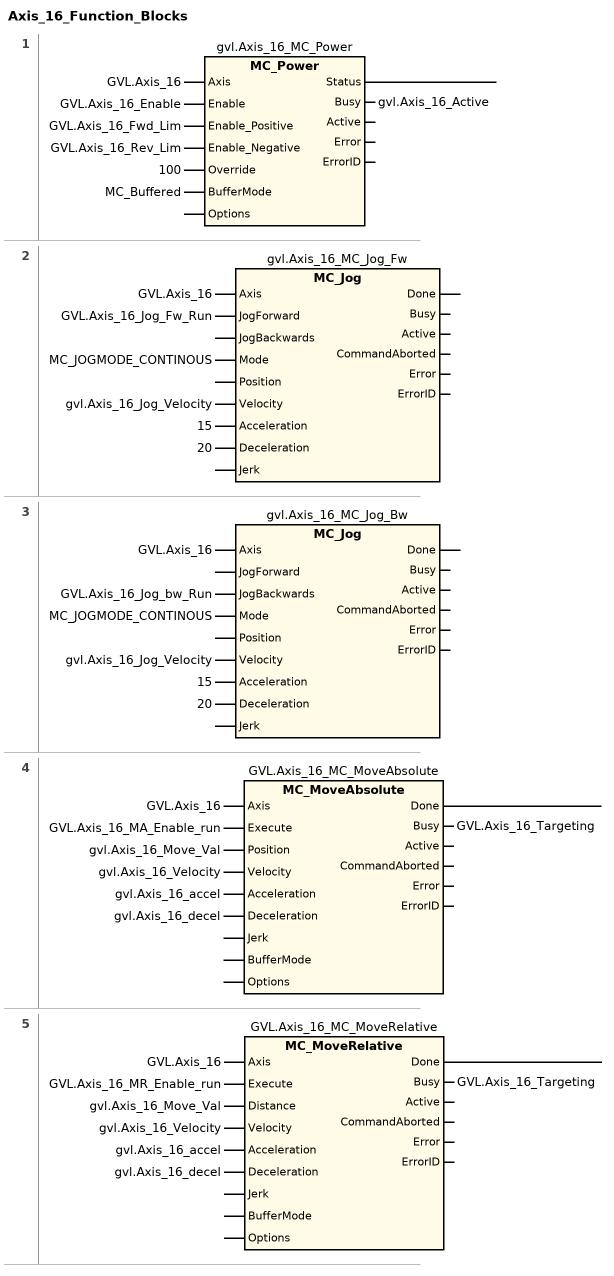
// NETWORK 1
gvl.Axis_16_MC_Power(
    Axis := GVL.Axis_16,
    Enable := GVL.Axis_16_Enable,
    Enable_Positive := GVL.Axis_16_Fwd_Lim,
    Enable_Negative := GVL.Axis_16_Rev_Lim,
    Override := 100,
    BufferMode := MC_Buffered,
    Busy => gvl.Axis_16_Active); // MC_Power

// NETWORK 2
gvl.Axis_16_MC_Jog_Fw(
    Axis := GVL.Axis_16,
    JogForward := GVL.Axis_16_Jog_Fw_Run,
    Mode := MC_JOGMODE_CONTINOUS,
    Velocity := gvl.Axis_16_Jog_Velocity,
    Acceleration := 15,
    Deceleration := 20); // MC_Jog

// NETWORK 3
gvl.Axis_16_MC_Jog_Bw(
    Axis := GVL.Axis_16,
    JogBackwards := GVL.Axis_16_Jog_bw_Run,
    Mode := MC_JOGMODE_CONTINOUS,
    Velocity := gvl.Axis_16_Jog_Velocity,
    Acceleration := 15,
    Deceleration := 20); // MC_Jog

// NETWORK 4
GVL.Axis_16_MC_MoveAbsolute(
    Axis := GVL.Axis_16,
    Execute := GVL.Axis_16_MA_Enable_run,
    Position := gvl.Axis_16_Move_Val,
    Velocity := gvl.Axis_16_Velocity,
    Acceleration := gvl.Axis_16_accel,
    Deceleration := gvl.Axis_16_decel,
    Busy => GVL.Axis_16_Targeting); // MC_MoveAbsolute

// NETWORK 5
GVL.Axis_16_MC_MoveRelative(
    Axis := GVL.Axis_16,
    Execute := GVL.Axis_16_MR_Enable_run,
    Distance := gvl.Axis_16_Move_Val,
    Velocity := gvl.Axis_16_Velocity,
    Acceleration := gvl.Axis_16_accel,
    Deceleration := gvl.Axis_16_decel,
    Busy => GVL.Axis_16_Targeting); // MC_MoveRelative

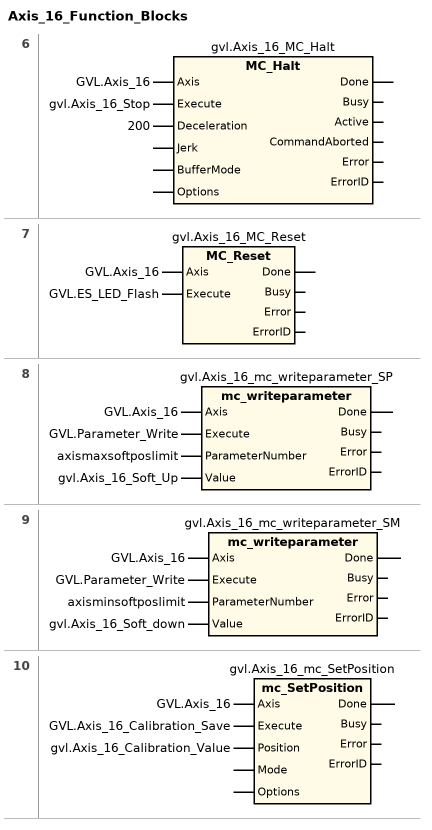
// NETWORK 6
gvl.Axis_16_MC_Halt(Axis := GVL.Axis_16, Execute := gvl.Axis_16_Stop, Deceleration := 200); // MC_Halt

// NETWORK 7
gvl.Axis_16_MC_Reset(Axis := GVL.Axis_16, Execute := GVL.ES_LED_Flash); // MC_Reset

// NETWORK 8
gvl.Axis_16_mc_writeparameter_SP(
    Axis := GVL.Axis_16,
    Execute := GVL.Parameter_Write,
    ParameterNumber := axismaxsoftposlimit,
    Value := gvl.Axis_16_Soft_Up); // mc_writeparameter

// NETWORK 9
gvl.Axis_16_mc_writeparameter_SM(
    Axis := GVL.Axis_16,
    Execute := GVL.Parameter_Write,
    ParameterNumber := axisminsoftposlimit,
    Value := gvl.Axis_16_Soft_down); // mc_writeparameter

// NETWORK 10
gvl.Axis_16_mc_SetPosition(
    Axis := GVL.Axis_16,
    Execute := GVL.Axis_16_Calibration_Save,
    Position := gvl.Axis_16_Calibration_Value); // mc_SetPosition

END_PROGRAM

// ---- POUs/Axis_16_Logic.TcPOU
PROGRAM Axis_16_Logic
VAR
	TON_0: TON;
	TON_1: TON;
	TON_2: TON;
	TON_3: TON;
	Axis_16_Velocity_Range: LREAL;
	Axis_16_Velocity_Scale: LREAL;
	Axis_16_Velocity_Raw: LREAL;
	Axis_16_Soft_Range: LREAL;
	Axis_16_Soft_Position: LREAL;
	Axis_16_Soft_Position_In_Range: LREAL;
END_VAR

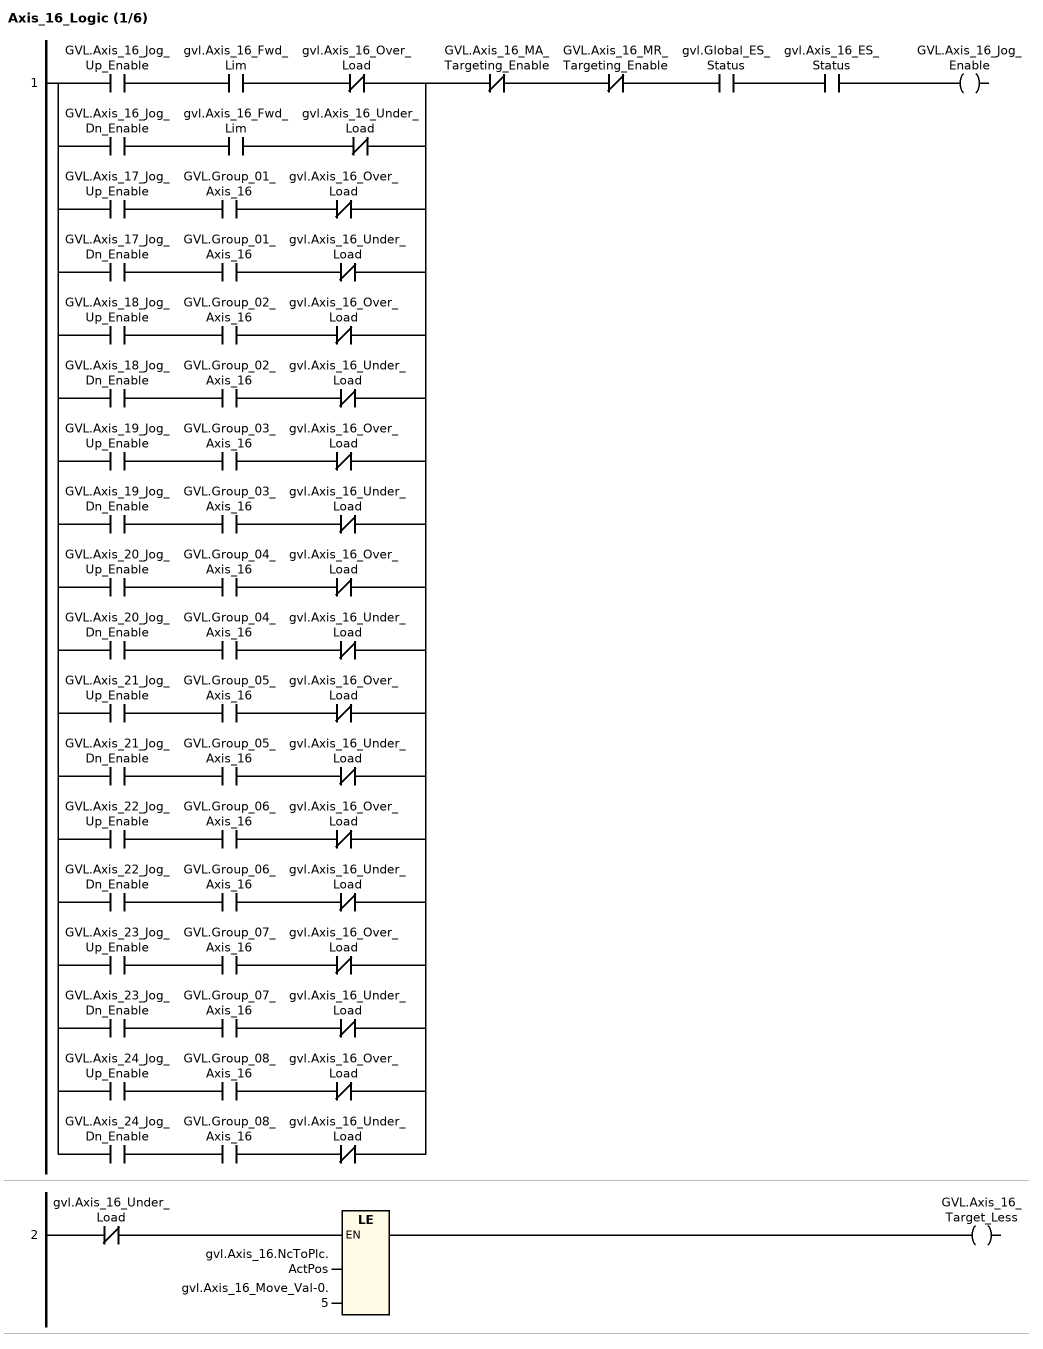
// NETWORK 1
GVL.Axis_16_Jog_Enable := (GVL.Axis_16_Jog_Up_Enable AND gvl.Axis_16_Fwd_Lim AND NOT gvl.Axis_16_Over_Load OR GVL.Axis_16_Jog_Dn_Enable AND gvl.Axis_16_Fwd_Lim AND NOT gvl.Axis_16_Under_Load OR GVL.Axis_17_Jog_Up_Enable AND GVL.Group_01_Axis_16 AND NOT gvl.Axis_16_Over_Load OR GVL.Axis_17_Jog_Dn_Enable AND GVL.Group_01_Axis_16 AND NOT gvl.Axis_16_Under_Load OR GVL.Axis_18_Jog_Up_Enable AND GVL.Group_02_Axis_16 AND NOT gvl.Axis_16_Over_Load OR GVL.Axis_18_Jog_Dn_Enable AND GVL.Group_02_Axis_16 AND NOT gvl.Axis_16_Under_Load OR GVL.Axis_19_Jog_Up_Enable AND GVL.Group_03_Axis_16 AND NOT gvl.Axis_16_Over_Load OR GVL.Axis_19_Jog_Dn_Enable AND GVL.Group_03_Axis_16 AND NOT gvl.Axis_16_Under_Load OR GVL.Axis_20_Jog_Up_Enable AND GVL.Group_04_Axis_16 AND NOT gvl.Axis_16_Over_Load OR GVL.Axis_20_Jog_Dn_Enable AND GVL.Group_04_Axis_16 AND NOT gvl.Axis_16_Under_Load OR GVL.Axis_21_Jog_Up_Enable AND GVL.Group_05_Axis_16 AND NOT gvl.Axis_16_Over_Load OR GVL.Axis_21_Jog_Dn_Enable AND GVL.Group_05_Axis_16 AND NOT gvl.Axis_16_Under_Load OR GVL.Axis_22_Jog_Up_Enable AND GVL.Group_06_Axis_16 AND NOT gvl.Axis_16_Over_Load OR GVL.Axis_22_Jog_Dn_Enable AND GVL.Group_06_Axis_16 AND NOT gvl.Axis_16_Under_Load OR GVL.Axis_23_Jog_Up_Enable AND GVL.Group_07_Axis_16 AND NOT gvl.Axis_16_Over_Load OR GVL.Axis_23_Jog_Dn_Enable AND GVL.Group_07_Axis_16 AND NOT gvl.Axis_16_Under_Load OR GVL.Axis_24_Jog_Up_Enable AND GVL.Group_08_Axis_16 AND NOT gvl.Axis_16_Over_Load OR GVL.Axis_24_Jog_Dn_Enable AND GVL.Group_08_Axis_16 AND NOT gvl.Axis_16_Under_Load) AND NOT GVL.Axis_16_MA_Targeting_Enable AND NOT GVL.Axis_16_MR_Targeting_Enable AND gvl.Global_ES_Status AND gvl.Axis_16_ES_Status;

// NETWORK 2
GVL.Axis_16_Target_Less := NOT gvl.Axis_16_Under_Load AND gvl.Axis_16.NcToPlc.ActPos <= (gvl.Axis_16_Move_Val-0.5);

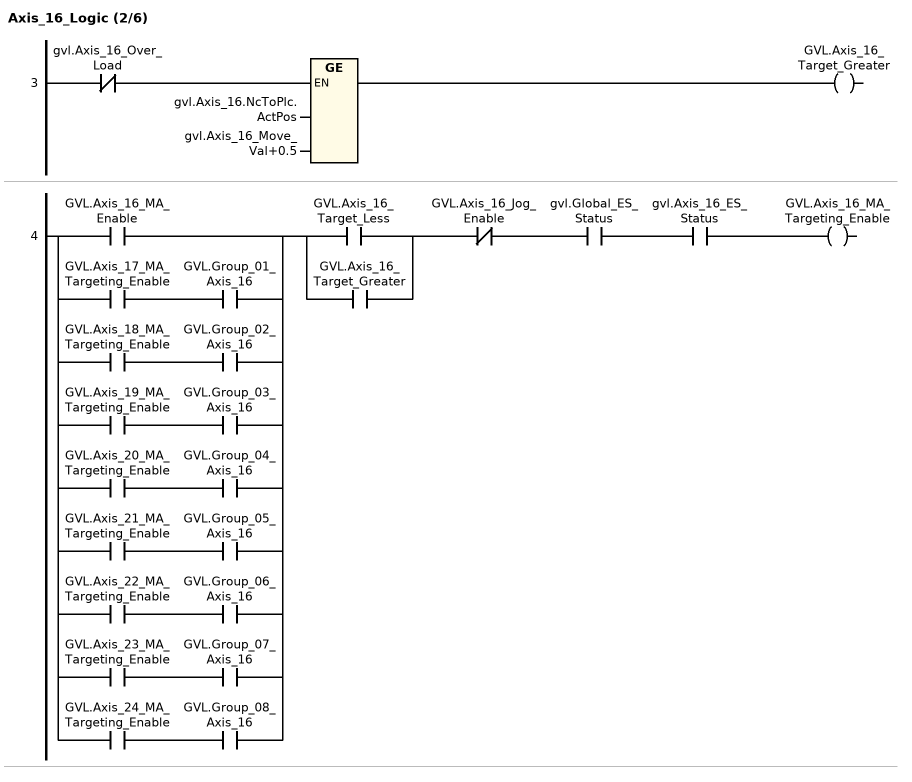
// NETWORK 3
GVL.Axis_16_Target_Greater := NOT gvl.Axis_16_Over_Load AND gvl.Axis_16.NcToPlc.ActPos >= (gvl.Axis_16_Move_Val+0.5);

// NETWORK 4
GVL.Axis_16_MA_Targeting_Enable := (GVL.Axis_16_MA_Enable OR GVL.Axis_17_MA_Targeting_Enable AND GVL.Group_01_Axis_16 OR GVL.Axis_18_MA_Targeting_Enable AND GVL.Group_02_Axis_16 OR GVL.Axis_19_MA_Targeting_Enable AND GVL.Group_03_Axis_16 OR GVL.Axis_20_MA_Targeting_Enable AND GVL.Group_04_Axis_16 OR GVL.Axis_21_MA_Targeting_Enable AND GVL.Group_05_Axis_16 OR GVL.Axis_22_MA_Targeting_Enable AND GVL.Group_06_Axis_16 OR GVL.Axis_23_MA_Targeting_Enable AND GVL.Group_07_Axis_16 OR GVL.Axis_24_MA_Targeting_Enable AND GVL.Group_08_Axis_16) AND (GVL.Axis_16_Target_Less OR GVL.Axis_16_Target_Greater) AND NOT GVL.Axis_16_Jog_Enable AND gvl.Global_ES_Status AND gvl.Axis_16_ES_Status;

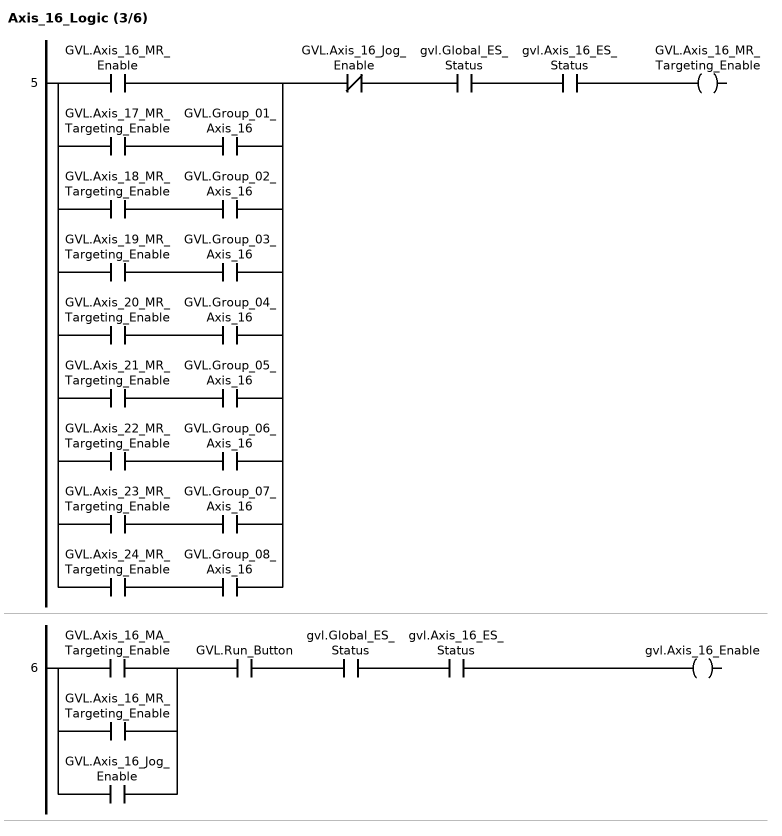
// NETWORK 5
GVL.Axis_16_MR_Targeting_Enable := (GVL.Axis_16_MR_Enable OR GVL.Axis_17_MR_Targeting_Enable AND GVL.Group_01_Axis_16 OR GVL.Axis_18_MR_Targeting_Enable AND GVL.Group_02_Axis_16 OR GVL.Axis_19_MR_Targeting_Enable AND GVL.Group_03_Axis_16 OR GVL.Axis_20_MR_Targeting_Enable AND GVL.Group_04_Axis_16 OR GVL.Axis_21_MR_Targeting_Enable AND GVL.Group_05_Axis_16 OR GVL.Axis_22_MR_Targeting_Enable AND GVL.Group_06_Axis_16 OR GVL.Axis_23_MR_Targeting_Enable AND GVL.Group_07_Axis_16 OR GVL.Axis_24_MR_Targeting_Enable AND GVL.Group_08_Axis_16) AND NOT GVL.Axis_16_Jog_Enable AND gvl.Global_ES_Status AND gvl.Axis_16_ES_Status;

// NETWORK 6
gvl.Axis_16_Enable := (GVL.Axis_16_MA_Targeting_Enable OR GVL.Axis_16_MR_Targeting_Enable OR GVL.Axis_16_Jog_Enable) AND GVL.Run_Button AND gvl.Global_ES_Status AND gvl.Axis_16_ES_Status;

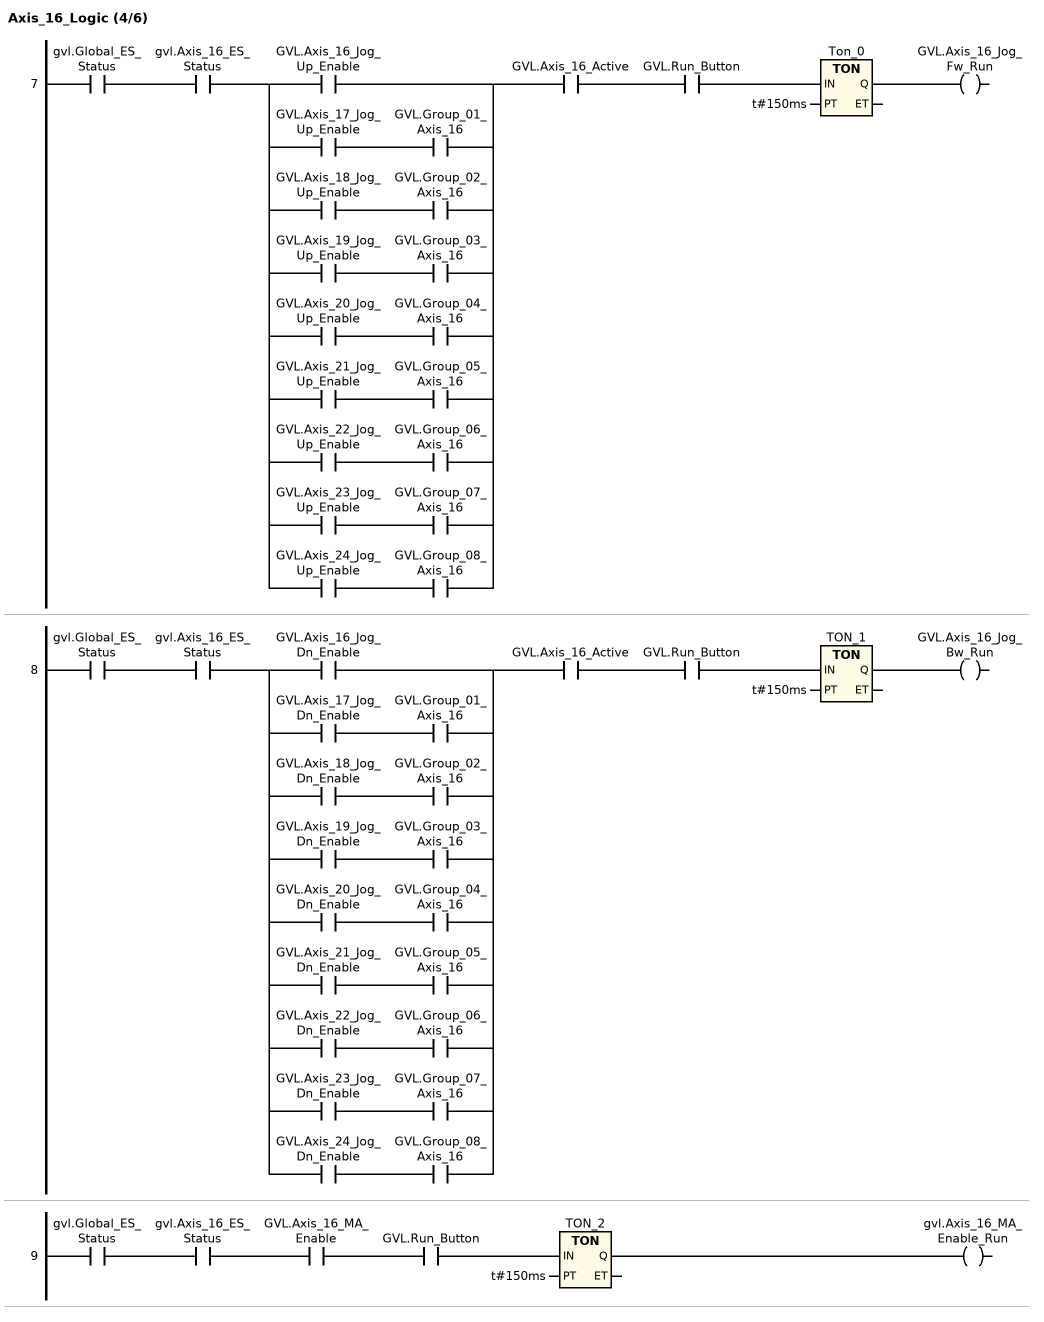
// NETWORK 7
Ton_0(IN := gvl.Global_ES_Status AND gvl.Axis_16_ES_Status AND (GVL.Axis_16_Jog_Up_Enable OR GVL.Axis_17_Jog_Up_Enable AND GVL.Group_01_Axis_16 OR GVL.Axis_18_Jog_Up_Enable AND GVL.Group_02_Axis_16 OR GVL.Axis_19_Jog_Up_Enable AND GVL.Group_03_Axis_16 OR GVL.Axis_20_Jog_Up_Enable AND GVL.Group_04_Axis_16 OR GVL.Axis_21_Jog_Up_Enable AND GVL.Group_05_Axis_16 OR GVL.Axis_22_Jog_Up_Enable AND GVL.Group_06_Axis_16 OR GVL.Axis_23_Jog_Up_Enable AND GVL.Group_07_Axis_16 OR GVL.Axis_24_Jog_Up_Enable AND GVL.Group_08_Axis_16) AND GVL.Axis_16_Active AND GVL.Run_Button, PT := t#150ms); // TON
GVL.Axis_16_Jog_Fw_Run := Ton_0.Q;

// NETWORK 8
TON_1(IN := gvl.Global_ES_Status AND gvl.Axis_16_ES_Status AND (GVL.Axis_16_Jog_Dn_Enable OR GVL.Axis_17_Jog_Dn_Enable AND GVL.Group_01_Axis_16 OR GVL.Axis_18_Jog_Dn_Enable AND GVL.Group_02_Axis_16 OR GVL.Axis_19_Jog_Dn_Enable AND GVL.Group_03_Axis_16 OR GVL.Axis_20_Jog_Dn_Enable AND GVL.Group_04_Axis_16 OR GVL.Axis_21_Jog_Dn_Enable AND GVL.Group_05_Axis_16 OR GVL.Axis_22_Jog_Dn_Enable AND GVL.Group_06_Axis_16 OR GVL.Axis_23_Jog_Dn_Enable AND GVL.Group_07_Axis_16 OR GVL.Axis_24_Jog_Dn_Enable AND GVL.Group_08_Axis_16) AND GVL.Axis_16_Active AND GVL.Run_Button, PT := t#150ms); // TON
GVL.Axis_16_Jog_Bw_Run := TON_1.Q;

// NETWORK 9
TON_2(IN := gvl.Global_ES_Status AND gvl.Axis_16_ES_Status AND GVL.Axis_16_MA_Enable AND GVL.Run_Button, PT := t#150ms); // TON
gvl.Axis_16_MA_Enable_Run := TON_2.Q;

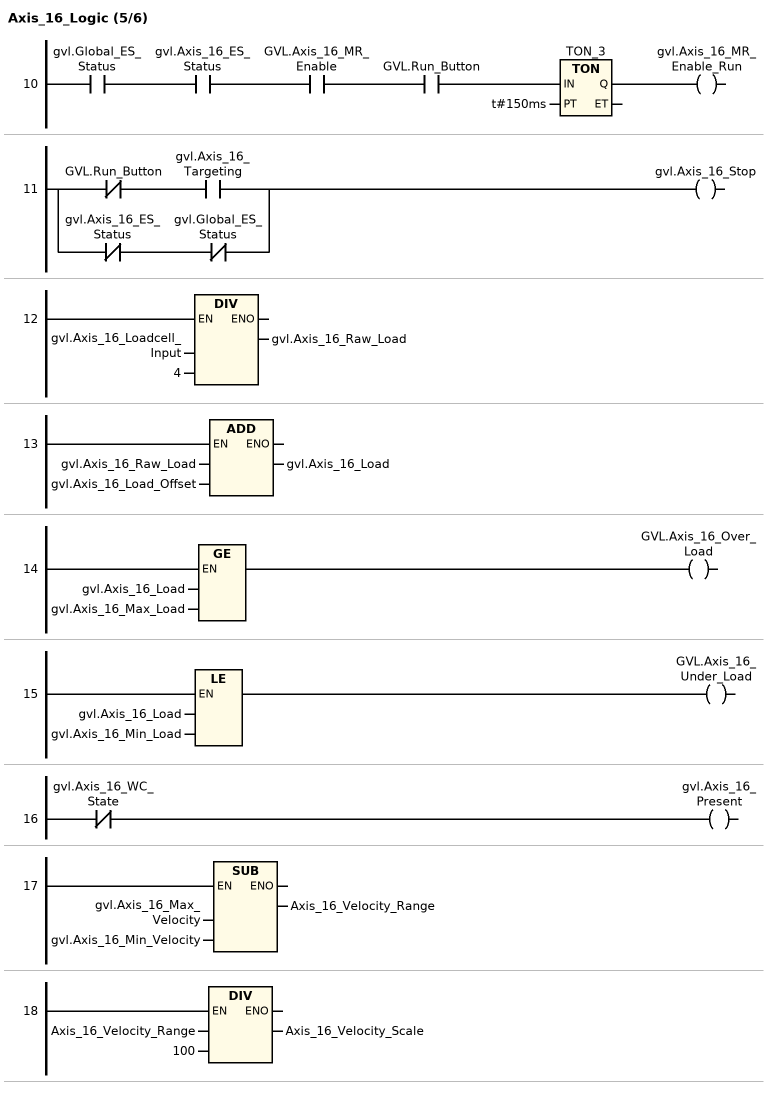
// NETWORK 10
TON_3(IN := gvl.Global_ES_Status AND gvl.Axis_16_ES_Status AND GVL.Axis_16_MR_Enable AND GVL.Run_Button, PT := t#150ms); // TON
gvl.Axis_16_MR_Enable_Run := TON_3.Q;

// NETWORK 11
gvl.Axis_16_Stop := NOT GVL.Run_Button AND gvl.Axis_16_Targeting OR NOT gvl.Axis_16_ES_Status AND NOT gvl.Global_ES_Status;

// NETWORK 12
gvl.Axis_16_Raw_Load := gvl.Axis_16_Loadcell_Input / 4;

// NETWORK 13
gvl.Axis_16_Load := gvl.Axis_16_Raw_Load + gvl.Axis_16_Load_Offset;

// NETWORK 14
GVL.Axis_16_Over_Load := gvl.Axis_16_Load >= gvl.Axis_16_Max_Load;

// NETWORK 15
GVL.Axis_16_Under_Load := gvl.Axis_16_Load <= gvl.Axis_16_Min_Load;

// NETWORK 16
gvl.Axis_16_Present := NOT gvl.Axis_16_WC_State;

// NETWORK 17
Axis_16_Velocity_Range := gvl.Axis_16_Max_Velocity - gvl.Axis_16_Min_Velocity;

// NETWORK 18
Axis_16_Velocity_Scale := Axis_16_Velocity_Range / 100;

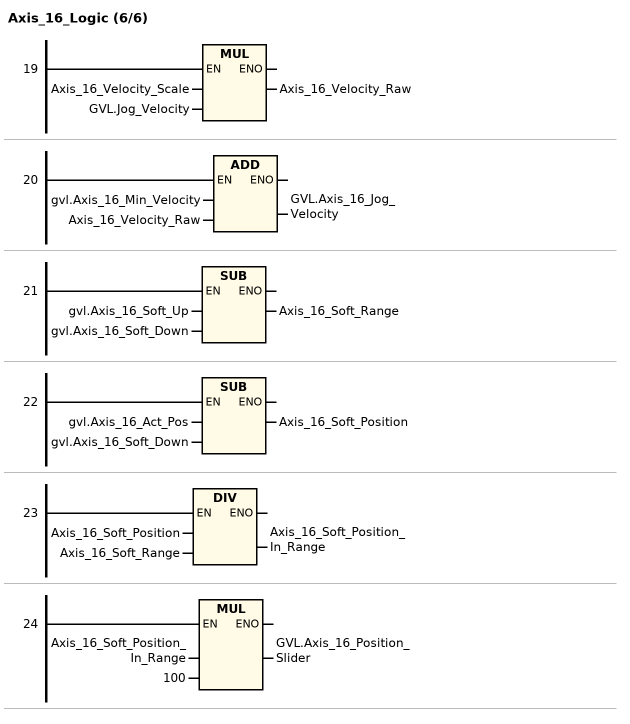
// NETWORK 19
Axis_16_Velocity_Raw := Axis_16_Velocity_Scale * GVL.Jog_Velocity;

// NETWORK 20
GVL.Axis_16_Jog_Velocity := gvl.Axis_16_Min_Velocity + Axis_16_Velocity_Raw;

// NETWORK 21
Axis_16_Soft_Range := gvl.Axis_16_Soft_Up - gvl.Axis_16_Soft_Down;

// NETWORK 22
Axis_16_Soft_Position := gvl.Axis_16_Act_Pos - gvl.Axis_16_Soft_Down;

// NETWORK 23
Axis_16_Soft_Position_In_Range := Axis_16_Soft_Position / Axis_16_Soft_Range;

// NETWORK 24
GVL.Axis_16_Position_Slider := Axis_16_Soft_Position_In_Range * 100;

END_PROGRAM

// ---- POUs/Group_01_Function_Blocks.TcPOU
PROGRAM Group_01_Function_Blocks
VAR
END_VAR

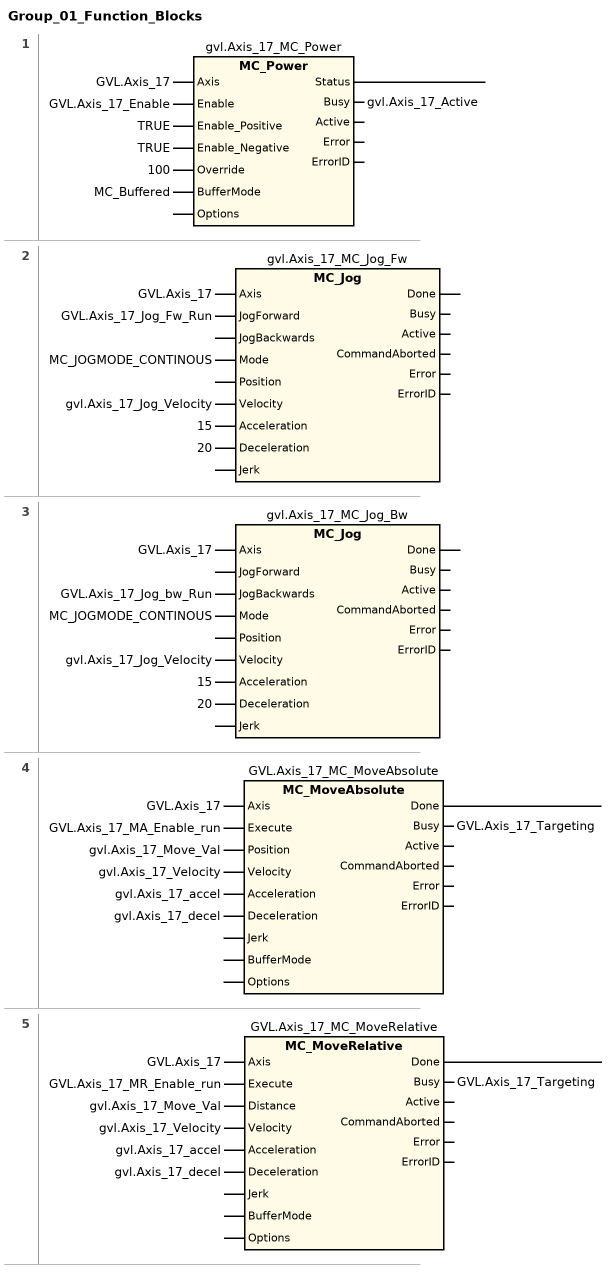
// NETWORK 1
gvl.Axis_17_MC_Power(
    Axis := GVL.Axis_17,
    Enable := GVL.Axis_17_Enable,
    Enable_Positive := TRUE,
    Enable_Negative := TRUE,
    Override := 100,
    BufferMode := MC_Buffered,
    Busy => gvl.Axis_17_Active); // MC_Power

// NETWORK 2
gvl.Axis_17_MC_Jog_Fw(
    Axis := GVL.Axis_17,
    JogForward := GVL.Axis_17_Jog_Fw_Run,
    Mode := MC_JOGMODE_CONTINOUS,
    Velocity := gvl.Axis_17_Jog_Velocity,
    Acceleration := 15,
    Deceleration := 20); // MC_Jog

// NETWORK 3
gvl.Axis_17_MC_Jog_Bw(
    Axis := GVL.Axis_17,
    JogBackwards := GVL.Axis_17_Jog_bw_Run,
    Mode := MC_JOGMODE_CONTINOUS,
    Velocity := gvl.Axis_17_Jog_Velocity,
    Acceleration := 15,
    Deceleration := 20); // MC_Jog

// NETWORK 4
GVL.Axis_17_MC_MoveAbsolute(
    Axis := GVL.Axis_17,
    Execute := GVL.Axis_17_MA_Enable_run,
    Position := gvl.Axis_17_Move_Val,
    Velocity := gvl.Axis_17_Velocity,
    Acceleration := gvl.Axis_17_accel,
    Deceleration := gvl.Axis_17_decel,
    Busy => GVL.Axis_17_Targeting); // MC_MoveAbsolute

// NETWORK 5
GVL.Axis_17_MC_MoveRelative(
    Axis := GVL.Axis_17,
    Execute := GVL.Axis_17_MR_Enable_run,
    Distance := gvl.Axis_17_Move_Val,
    Velocity := gvl.Axis_17_Velocity,
    Acceleration := gvl.Axis_17_accel,
    Deceleration := gvl.Axis_17_decel,
    Busy => GVL.Axis_17_Targeting); // MC_MoveRelative

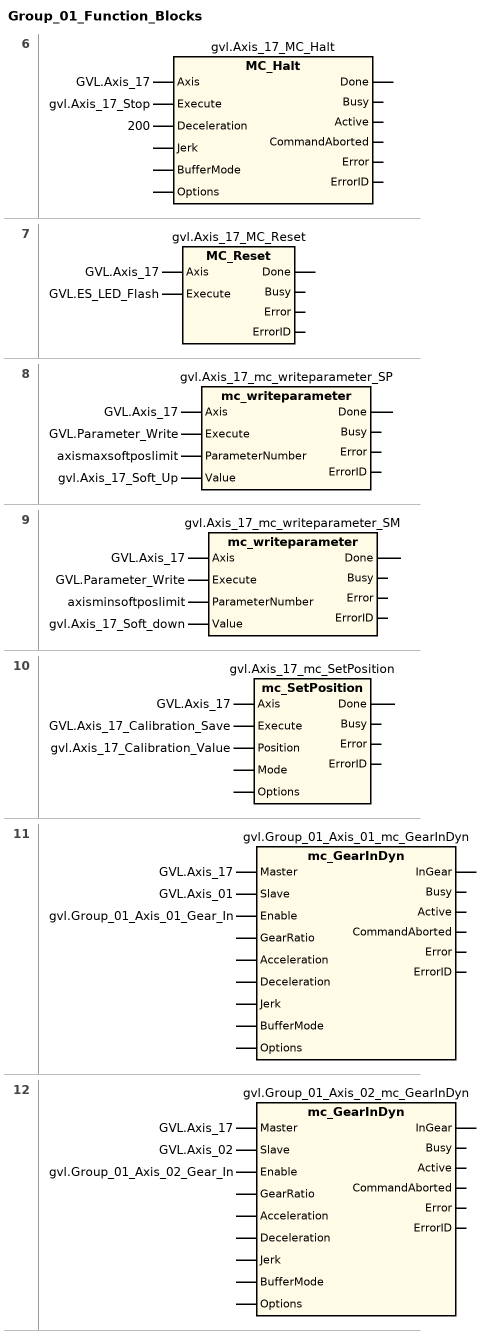
// NETWORK 6
gvl.Axis_17_MC_Halt(Axis := GVL.Axis_17, Execute := gvl.Axis_17_Stop, Deceleration := 200); // MC_Halt

// NETWORK 7
gvl.Axis_17_MC_Reset(Axis := GVL.Axis_17, Execute := GVL.ES_LED_Flash); // MC_Reset

// NETWORK 8
gvl.Axis_17_mc_writeparameter_SP(
    Axis := GVL.Axis_17,
    Execute := GVL.Parameter_Write,
    ParameterNumber := axismaxsoftposlimit,
    Value := gvl.Axis_17_Soft_Up); // mc_writeparameter

// NETWORK 9
gvl.Axis_17_mc_writeparameter_SM(
    Axis := GVL.Axis_17,
    Execute := GVL.Parameter_Write,
    ParameterNumber := axisminsoftposlimit,
    Value := gvl.Axis_17_Soft_down); // mc_writeparameter

// NETWORK 10
gvl.Axis_17_mc_SetPosition(
    Axis := GVL.Axis_17,
    Execute := GVL.Axis_17_Calibration_Save,
    Position := gvl.Axis_17_Calibration_Value); // mc_SetPosition

// NETWORK 11
gvl.Group_01_Axis_01_mc_GearInDyn(
    Master := GVL.Axis_17,
    Slave := GVL.Axis_01,
    Enable := gvl.Group_01_Axis_01_Gear_In); // mc_GearInDyn

// NETWORK 12
gvl.Group_01_Axis_02_mc_GearInDyn(
    Master := GVL.Axis_17,
    Slave := GVL.Axis_02,
    Enable := gvl.Group_01_Axis_02_Gear_In); // mc_GearInDyn

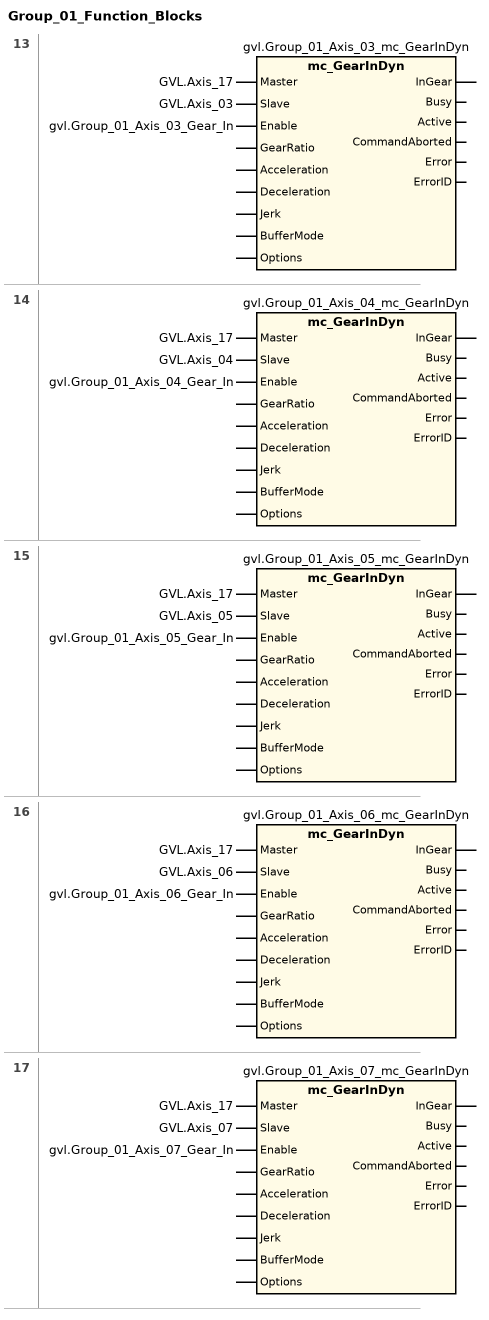
// NETWORK 13
gvl.Group_01_Axis_03_mc_GearInDyn(
    Master := GVL.Axis_17,
    Slave := GVL.Axis_03,
    Enable := gvl.Group_01_Axis_03_Gear_In); // mc_GearInDyn

// NETWORK 14
gvl.Group_01_Axis_04_mc_GearInDyn(
    Master := GVL.Axis_17,
    Slave := GVL.Axis_04,
    Enable := gvl.Group_01_Axis_04_Gear_In); // mc_GearInDyn

// NETWORK 15
gvl.Group_01_Axis_05_mc_GearInDyn(
    Master := GVL.Axis_17,
    Slave := GVL.Axis_05,
    Enable := gvl.Group_01_Axis_05_Gear_In); // mc_GearInDyn

// NETWORK 16
gvl.Group_01_Axis_06_mc_GearInDyn(
    Master := GVL.Axis_17,
    Slave := GVL.Axis_06,
    Enable := gvl.Group_01_Axis_06_Gear_In); // mc_GearInDyn

// NETWORK 17
gvl.Group_01_Axis_07_mc_GearInDyn(
    Master := GVL.Axis_17,
    Slave := GVL.Axis_07,
    Enable := gvl.Group_01_Axis_07_Gear_In); // mc_GearInDyn

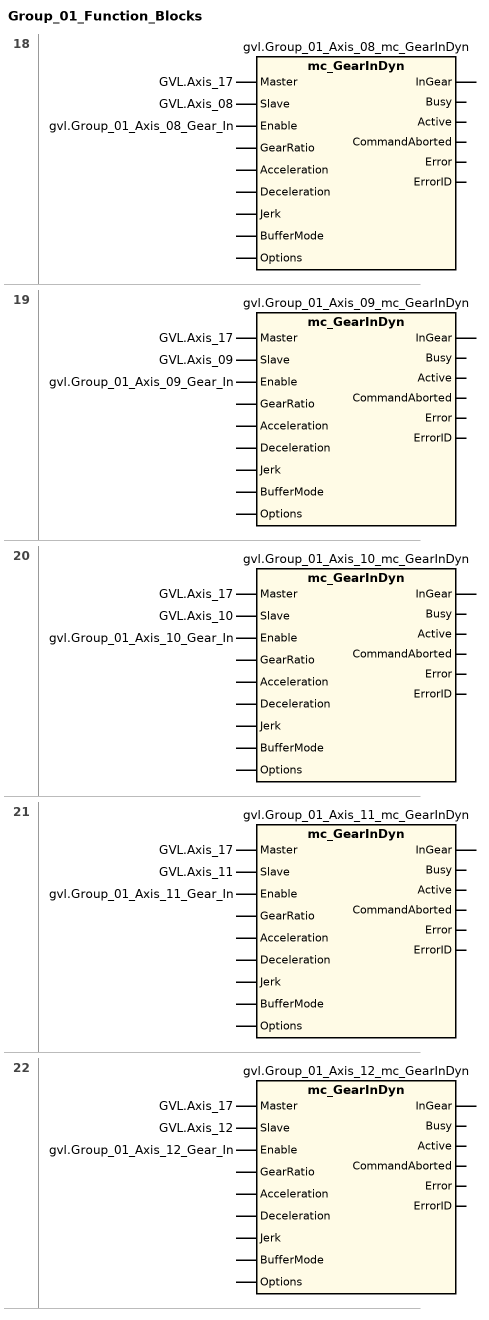
// NETWORK 18
gvl.Group_01_Axis_08_mc_GearInDyn(
    Master := GVL.Axis_17,
    Slave := GVL.Axis_08,
    Enable := gvl.Group_01_Axis_08_Gear_In); // mc_GearInDyn

// NETWORK 19
gvl.Group_01_Axis_09_mc_GearInDyn(
    Master := GVL.Axis_17,
    Slave := GVL.Axis_09,
    Enable := gvl.Group_01_Axis_09_Gear_In); // mc_GearInDyn

// NETWORK 20
gvl.Group_01_Axis_10_mc_GearInDyn(
    Master := GVL.Axis_17,
    Slave := GVL.Axis_10,
    Enable := gvl.Group_01_Axis_10_Gear_In); // mc_GearInDyn

// NETWORK 21
gvl.Group_01_Axis_11_mc_GearInDyn(
    Master := GVL.Axis_17,
    Slave := GVL.Axis_11,
    Enable := gvl.Group_01_Axis_11_Gear_In); // mc_GearInDyn

// NETWORK 22
gvl.Group_01_Axis_12_mc_GearInDyn(
    Master := GVL.Axis_17,
    Slave := GVL.Axis_12,
    Enable := gvl.Group_01_Axis_12_Gear_In); // mc_GearInDyn

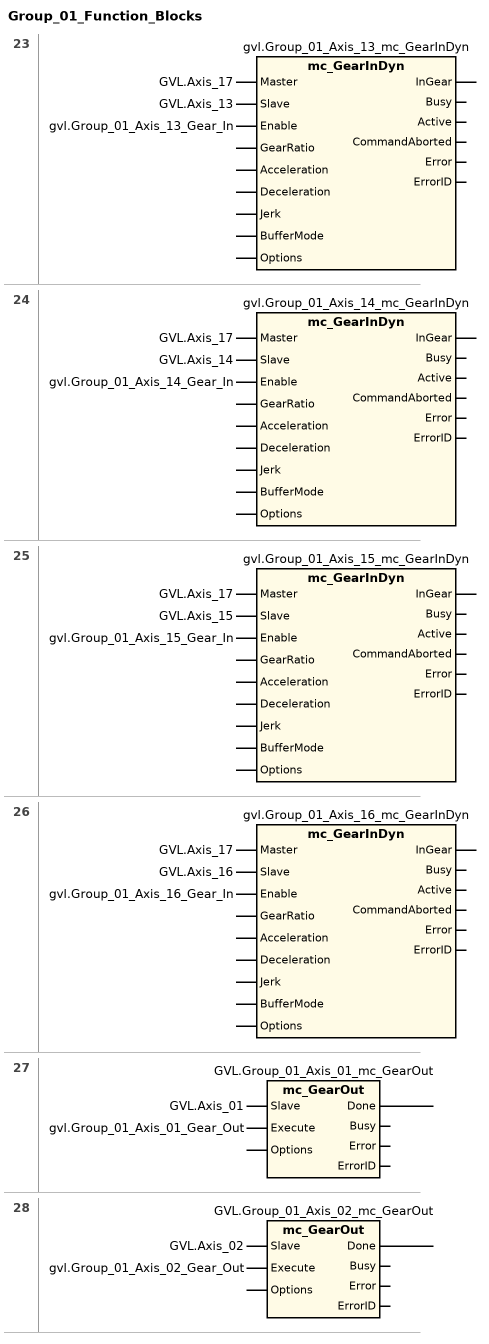
// NETWORK 23
gvl.Group_01_Axis_13_mc_GearInDyn(
    Master := GVL.Axis_17,
    Slave := GVL.Axis_13,
    Enable := gvl.Group_01_Axis_13_Gear_In); // mc_GearInDyn

// NETWORK 24
gvl.Group_01_Axis_14_mc_GearInDyn(
    Master := GVL.Axis_17,
    Slave := GVL.Axis_14,
    Enable := gvl.Group_01_Axis_14_Gear_In); // mc_GearInDyn

// NETWORK 25
gvl.Group_01_Axis_15_mc_GearInDyn(
    Master := GVL.Axis_17,
    Slave := GVL.Axis_15,
    Enable := gvl.Group_01_Axis_15_Gear_In); // mc_GearInDyn

// NETWORK 26
gvl.Group_01_Axis_16_mc_GearInDyn(
    Master := GVL.Axis_17,
    Slave := GVL.Axis_16,
    Enable := gvl.Group_01_Axis_16_Gear_In); // mc_GearInDyn

// NETWORK 27
GVL.Group_01_Axis_01_mc_GearOut(Slave := GVL.Axis_01, Execute := gvl.Group_01_Axis_01_Gear_Out); // mc_GearOut

// NETWORK 28
GVL.Group_01_Axis_02_mc_GearOut(Slave := GVL.Axis_02, Execute := gvl.Group_01_Axis_02_Gear_Out); // mc_GearOut

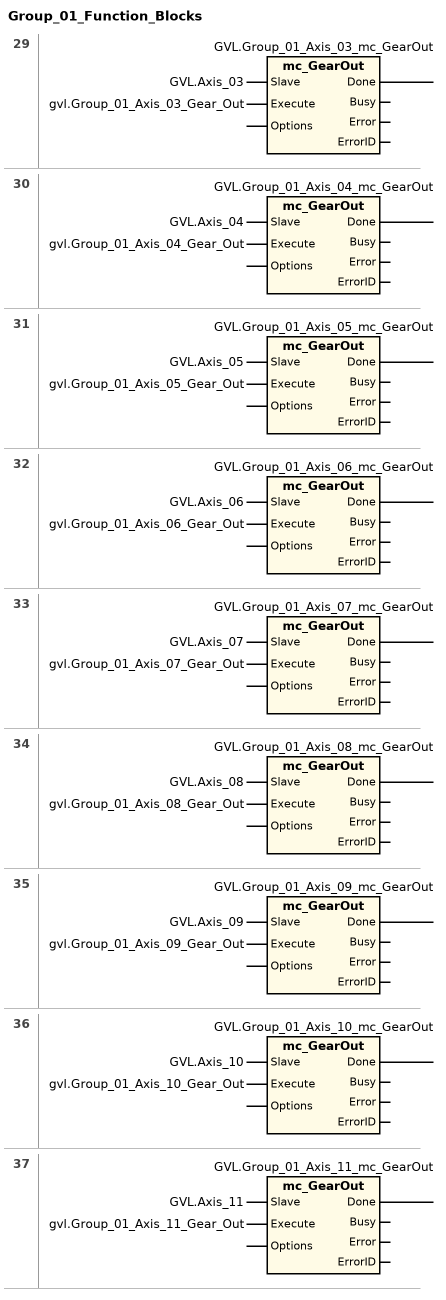
// NETWORK 29
GVL.Group_01_Axis_03_mc_GearOut(Slave := GVL.Axis_03, Execute := gvl.Group_01_Axis_03_Gear_Out); // mc_GearOut

// NETWORK 30
GVL.Group_01_Axis_04_mc_GearOut(Slave := GVL.Axis_04, Execute := gvl.Group_01_Axis_04_Gear_Out); // mc_GearOut

// NETWORK 31
GVL.Group_01_Axis_05_mc_GearOut(Slave := GVL.Axis_05, Execute := gvl.Group_01_Axis_05_Gear_Out); // mc_GearOut

// NETWORK 32
GVL.Group_01_Axis_06_mc_GearOut(Slave := GVL.Axis_06, Execute := gvl.Group_01_Axis_06_Gear_Out); // mc_GearOut

// NETWORK 33
GVL.Group_01_Axis_07_mc_GearOut(Slave := GVL.Axis_07, Execute := gvl.Group_01_Axis_07_Gear_Out); // mc_GearOut

// NETWORK 34
GVL.Group_01_Axis_08_mc_GearOut(Slave := GVL.Axis_08, Execute := gvl.Group_01_Axis_08_Gear_Out); // mc_GearOut

// NETWORK 35
GVL.Group_01_Axis_09_mc_GearOut(Slave := GVL.Axis_09, Execute := gvl.Group_01_Axis_09_Gear_Out); // mc_GearOut

// NETWORK 36
GVL.Group_01_Axis_10_mc_GearOut(Slave := GVL.Axis_10, Execute := gvl.Group_01_Axis_10_Gear_Out); // mc_GearOut

// NETWORK 37
GVL.Group_01_Axis_11_mc_GearOut(Slave := GVL.Axis_11, Execute := gvl.Group_01_Axis_11_Gear_Out); // mc_GearOut

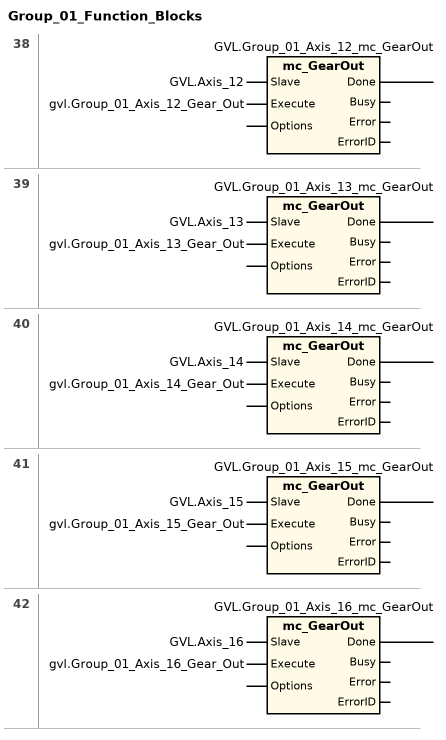
// NETWORK 38
GVL.Group_01_Axis_12_mc_GearOut(Slave := GVL.Axis_12, Execute := gvl.Group_01_Axis_12_Gear_Out); // mc_GearOut

// NETWORK 39
GVL.Group_01_Axis_13_mc_GearOut(Slave := GVL.Axis_13, Execute := gvl.Group_01_Axis_13_Gear_Out); // mc_GearOut

// NETWORK 40
GVL.Group_01_Axis_14_mc_GearOut(Slave := GVL.Axis_14, Execute := gvl.Group_01_Axis_14_Gear_Out); // mc_GearOut

// NETWORK 41
GVL.Group_01_Axis_15_mc_GearOut(Slave := GVL.Axis_15, Execute := gvl.Group_01_Axis_15_Gear_Out); // mc_GearOut

// NETWORK 42
GVL.Group_01_Axis_16_mc_GearOut(Slave := GVL.Axis_16, Execute := gvl.Group_01_Axis_16_Gear_Out); // mc_GearOut

END_PROGRAM

// ---- POUs/Group_01_Logic.TcPOU
PROGRAM Group_01_Logic
VAR
	TON_0: TON;
	TON_1: TON;
	TON_2: TON;
	TON_3: TON;
	
Axis_17_Velocity_Range: LREAL;
Axis_17_Velocity_Scale: LREAL;
Axis_17_Velocity_Raw: LREAL;
Axis_17_Soft_Range: LREAL;
Axis_17_Soft_Position: LREAL;
Axis_17_Soft_Position_In_Range: LREAL;
END_VAR
VAR // added by the converter: edge detectors and wires of the graphical bodies
    _w1, _w2, _w3, _w4, _w5, _w6, _w7, _w8, _w9, _w10, _w11, _w12, _w13, _w14, _w15, _w16, _w17, _w18, _w19, _w20, _w21, _w22, _w23, _w24, _w25, _w26, _w27, _w28, _w29, _w30, _w31, _w32 : BOOL;
END_VAR

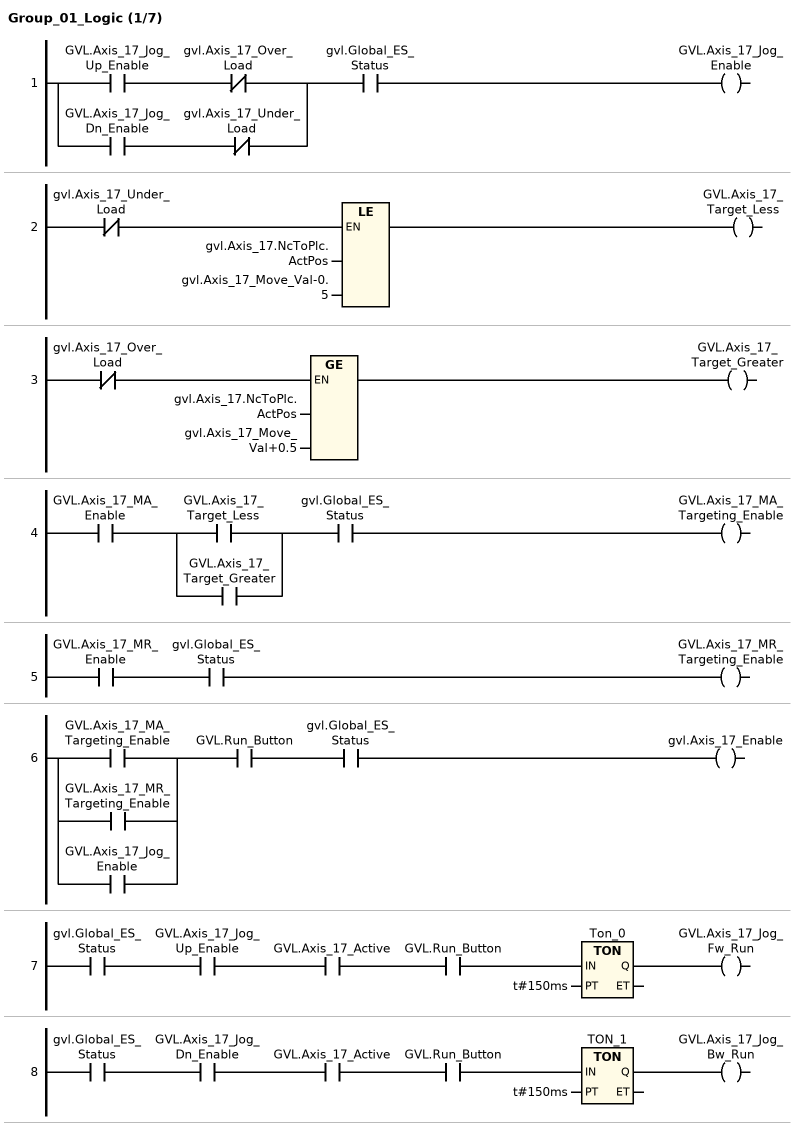
// NETWORK 1
GVL.Axis_17_Jog_Enable := (GVL.Axis_17_Jog_Up_Enable AND NOT gvl.Axis_17_Over_Load OR GVL.Axis_17_Jog_Dn_Enable AND NOT gvl.Axis_17_Under_Load) AND gvl.Global_ES_Status;

// NETWORK 2
GVL.Axis_17_Target_Less := NOT gvl.Axis_17_Under_Load AND gvl.Axis_17.NcToPlc.ActPos <= (gvl.Axis_17_Move_Val-0.5);

// NETWORK 3
GVL.Axis_17_Target_Greater := NOT gvl.Axis_17_Over_Load AND gvl.Axis_17.NcToPlc.ActPos >= (gvl.Axis_17_Move_Val+0.5);

// NETWORK 4
GVL.Axis_17_MA_Targeting_Enable := GVL.Axis_17_MA_Enable AND (GVL.Axis_17_Target_Less OR GVL.Axis_17_Target_Greater) AND gvl.Global_ES_Status;

// NETWORK 5
GVL.Axis_17_MR_Targeting_Enable := GVL.Axis_17_MR_Enable AND gvl.Global_ES_Status;

// NETWORK 6
gvl.Axis_17_Enable := (GVL.Axis_17_MA_Targeting_Enable OR GVL.Axis_17_MR_Targeting_Enable OR GVL.Axis_17_Jog_Enable) AND GVL.Run_Button AND gvl.Global_ES_Status;

// NETWORK 7
Ton_0(IN := gvl.Global_ES_Status AND GVL.Axis_17_Jog_Up_Enable AND GVL.Axis_17_Active AND GVL.Run_Button, PT := t#150ms); // TON
GVL.Axis_17_Jog_Fw_Run := Ton_0.Q;

// NETWORK 8
TON_1(IN := gvl.Global_ES_Status AND GVL.Axis_17_Jog_Dn_Enable AND GVL.Axis_17_Active AND GVL.Run_Button, PT := t#150ms); // TON
GVL.Axis_17_Jog_Bw_Run := TON_1.Q;

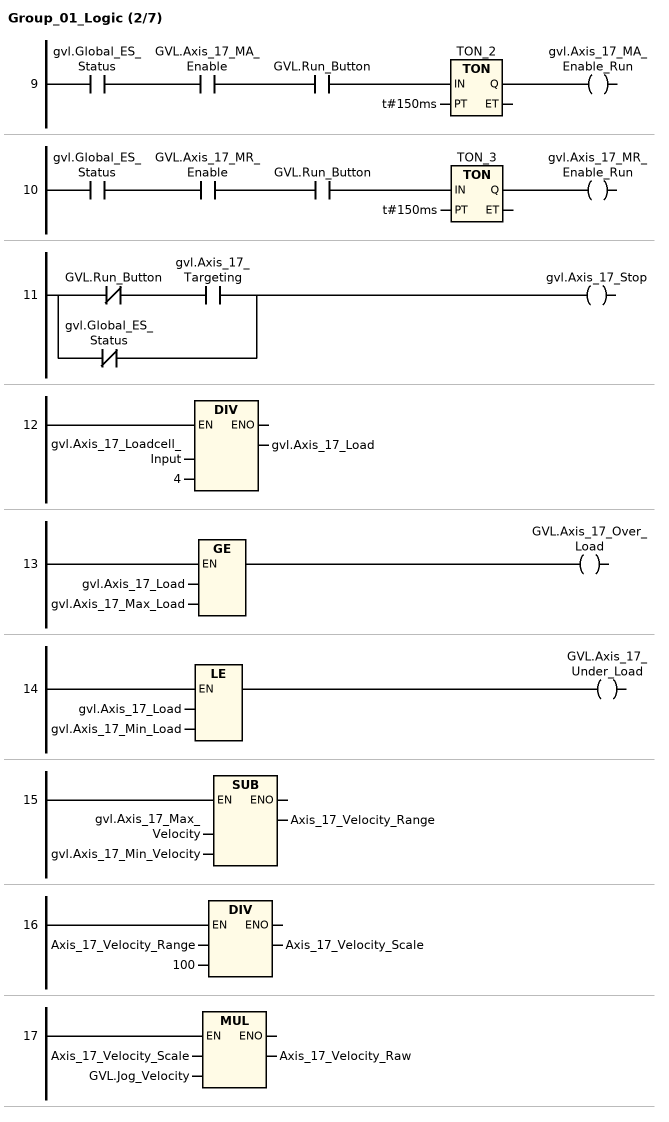
// NETWORK 9
TON_2(IN := gvl.Global_ES_Status AND GVL.Axis_17_MA_Enable AND GVL.Run_Button, PT := t#150ms); // TON
gvl.Axis_17_MA_Enable_Run := TON_2.Q;

// NETWORK 10
TON_3(IN := gvl.Global_ES_Status AND GVL.Axis_17_MR_Enable AND GVL.Run_Button, PT := t#150ms); // TON
gvl.Axis_17_MR_Enable_Run := TON_3.Q;

// NETWORK 11
gvl.Axis_17_Stop := NOT GVL.Run_Button AND gvl.Axis_17_Targeting OR NOT gvl.Global_ES_Status;

// NETWORK 12
gvl.Axis_17_Load := gvl.Axis_17_Loadcell_Input / 4;

// NETWORK 13
GVL.Axis_17_Over_Load := gvl.Axis_17_Load >= gvl.Axis_17_Max_Load;

// NETWORK 14
GVL.Axis_17_Under_Load := gvl.Axis_17_Load <= gvl.Axis_17_Min_Load;

// NETWORK 15
Axis_17_Velocity_Range := gvl.Axis_17_Max_Velocity - gvl.Axis_17_Min_Velocity;

// NETWORK 16
Axis_17_Velocity_Scale := Axis_17_Velocity_Range / 100;

// NETWORK 17
Axis_17_Velocity_Raw := Axis_17_Velocity_Scale * GVL.Jog_Velocity;

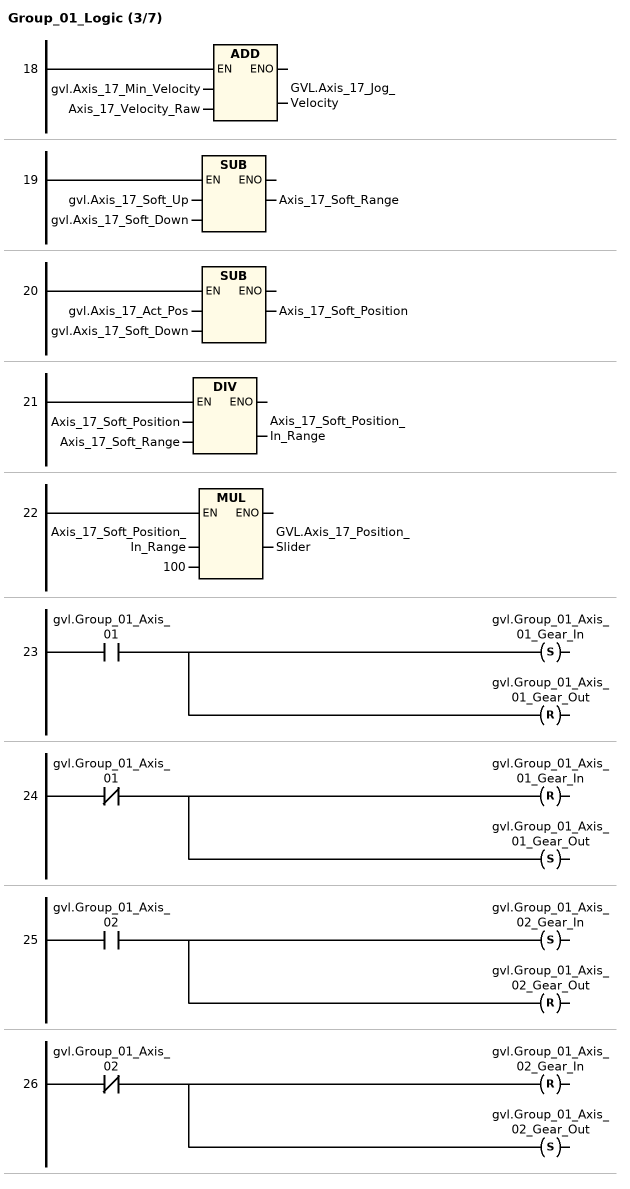
// NETWORK 18
GVL.Axis_17_Jog_Velocity := gvl.Axis_17_Min_Velocity + Axis_17_Velocity_Raw;

// NETWORK 19
Axis_17_Soft_Range := gvl.Axis_17_Soft_Up - gvl.Axis_17_Soft_Down;

// NETWORK 20
Axis_17_Soft_Position := gvl.Axis_17_Act_Pos - gvl.Axis_17_Soft_Down;

// NETWORK 21
Axis_17_Soft_Position_In_Range := Axis_17_Soft_Position / Axis_17_Soft_Range;

// NETWORK 22
GVL.Axis_17_Position_Slider := Axis_17_Soft_Position_In_Range * 100;

// NETWORK 23
_w1 := gvl.Group_01_Axis_01;
gvl.Group_01_Axis_01_Gear_In S= _w1;
gvl.Group_01_Axis_01_Gear_Out R= _w1;

// NETWORK 24
_w2 := NOT gvl.Group_01_Axis_01;
gvl.Group_01_Axis_01_Gear_In R= _w2;
gvl.Group_01_Axis_01_Gear_Out S= _w2;

// NETWORK 25
_w3 := gvl.Group_01_Axis_02;
gvl.Group_01_Axis_02_Gear_In S= _w3;
gvl.Group_01_Axis_02_Gear_Out R= _w3;

// NETWORK 26
_w4 := NOT gvl.Group_01_Axis_02;
gvl.Group_01_Axis_02_Gear_In R= _w4;
gvl.Group_01_Axis_02_Gear_Out S= _w4;

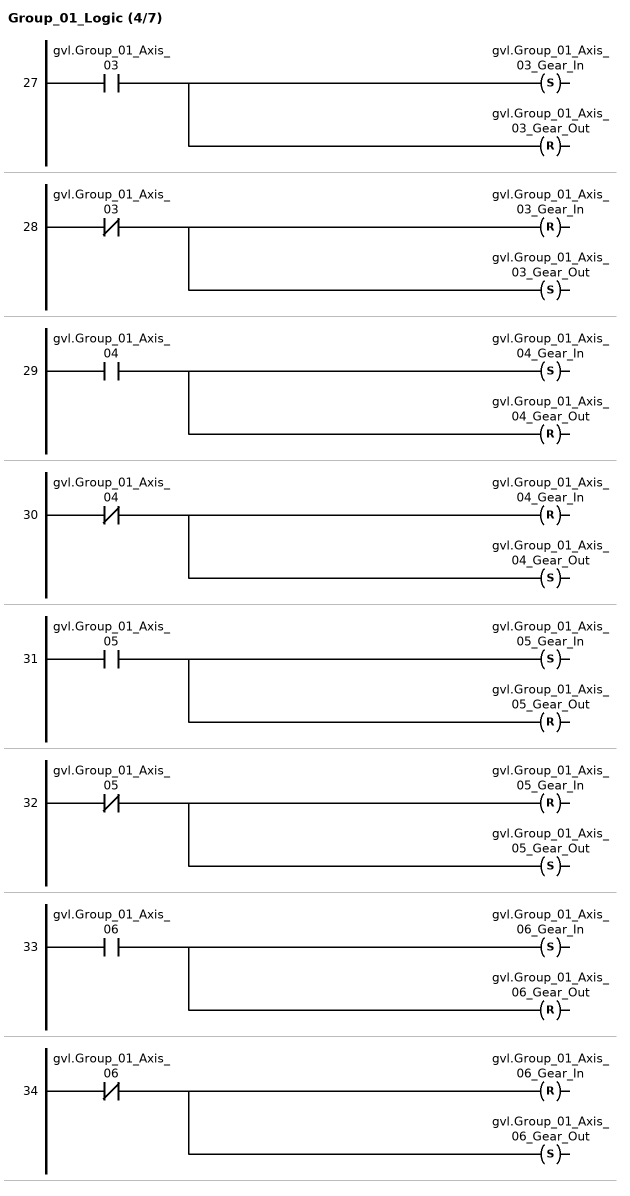
// NETWORK 27
_w5 := gvl.Group_01_Axis_03;
gvl.Group_01_Axis_03_Gear_In S= _w5;
gvl.Group_01_Axis_03_Gear_Out R= _w5;

// NETWORK 28
_w6 := NOT gvl.Group_01_Axis_03;
gvl.Group_01_Axis_03_Gear_In R= _w6;
gvl.Group_01_Axis_03_Gear_Out S= _w6;

// NETWORK 29
_w7 := gvl.Group_01_Axis_04;
gvl.Group_01_Axis_04_Gear_In S= _w7;
gvl.Group_01_Axis_04_Gear_Out R= _w7;

// NETWORK 30
_w8 := NOT gvl.Group_01_Axis_04;
gvl.Group_01_Axis_04_Gear_In R= _w8;
gvl.Group_01_Axis_04_Gear_Out S= _w8;

// NETWORK 31
_w9 := gvl.Group_01_Axis_05;
gvl.Group_01_Axis_05_Gear_In S= _w9;
gvl.Group_01_Axis_05_Gear_Out R= _w9;

// NETWORK 32
_w10 := NOT gvl.Group_01_Axis_05;
gvl.Group_01_Axis_05_Gear_In R= _w10;
gvl.Group_01_Axis_05_Gear_Out S= _w10;

// NETWORK 33
_w11 := gvl.Group_01_Axis_06;
gvl.Group_01_Axis_06_Gear_In S= _w11;
gvl.Group_01_Axis_06_Gear_Out R= _w11;

// NETWORK 34
_w12 := NOT gvl.Group_01_Axis_06;
gvl.Group_01_Axis_06_Gear_In R= _w12;
gvl.Group_01_Axis_06_Gear_Out S= _w12;

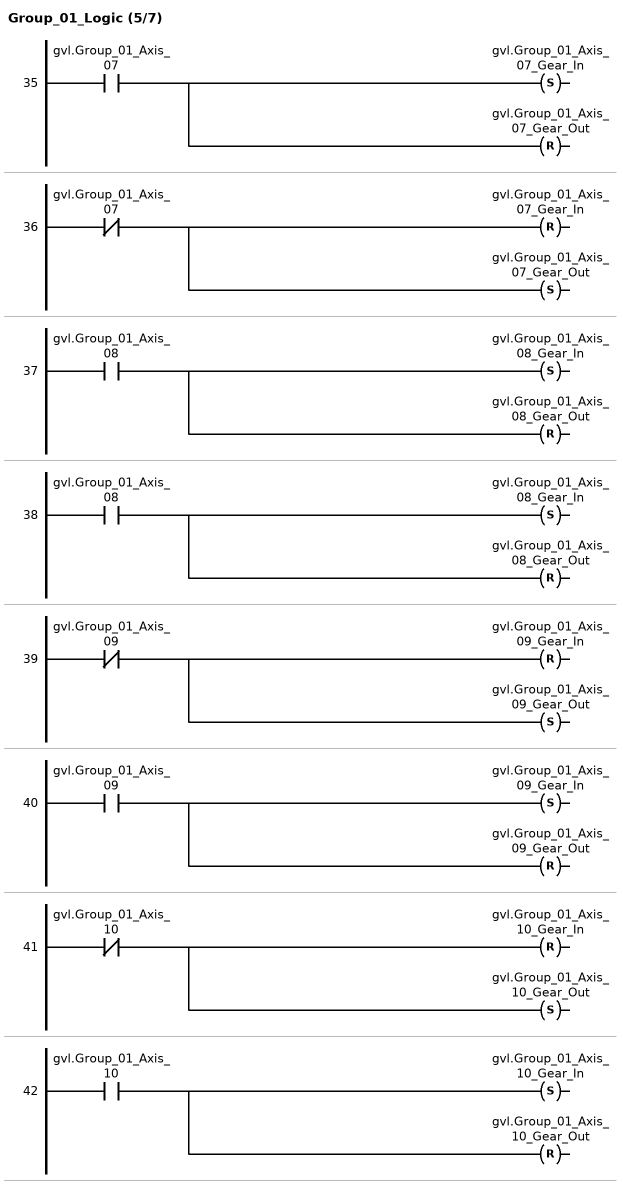
// NETWORK 35
_w13 := gvl.Group_01_Axis_07;
gvl.Group_01_Axis_07_Gear_In S= _w13;
gvl.Group_01_Axis_07_Gear_Out R= _w13;

// NETWORK 36
_w14 := NOT gvl.Group_01_Axis_07;
gvl.Group_01_Axis_07_Gear_In R= _w14;
gvl.Group_01_Axis_07_Gear_Out S= _w14;

// NETWORK 37
_w15 := gvl.Group_01_Axis_08;
gvl.Group_01_Axis_08_Gear_In S= _w15;
gvl.Group_01_Axis_08_Gear_Out R= _w15;

// NETWORK 38
_w16 := gvl.Group_01_Axis_08;
gvl.Group_01_Axis_08_Gear_In S= _w16;
gvl.Group_01_Axis_08_Gear_Out R= _w16;

// NETWORK 39
_w17 := NOT gvl.Group_01_Axis_09;
gvl.Group_01_Axis_09_Gear_In R= _w17;
gvl.Group_01_Axis_09_Gear_Out S= _w17;

// NETWORK 40
_w18 := gvl.Group_01_Axis_09;
gvl.Group_01_Axis_09_Gear_In S= _w18;
gvl.Group_01_Axis_09_Gear_Out R= _w18;

// NETWORK 41
_w19 := NOT gvl.Group_01_Axis_10;
gvl.Group_01_Axis_10_Gear_In R= _w19;
gvl.Group_01_Axis_10_Gear_Out S= _w19;

// NETWORK 42
_w20 := gvl.Group_01_Axis_10;
gvl.Group_01_Axis_10_Gear_In S= _w20;
gvl.Group_01_Axis_10_Gear_Out R= _w20;

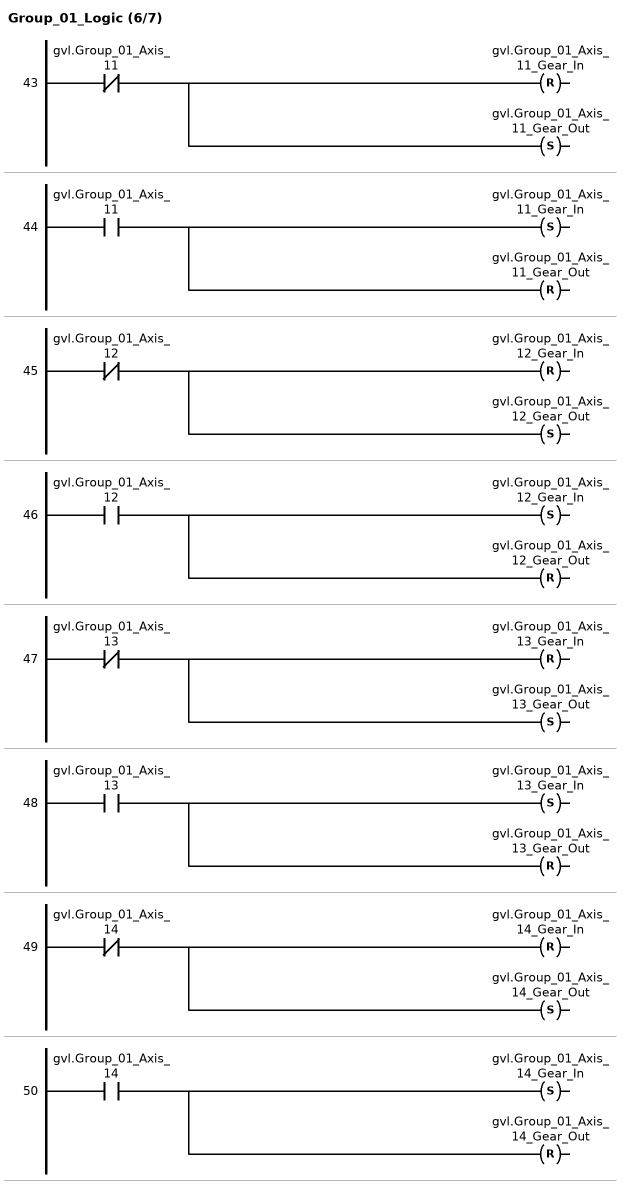
// NETWORK 43
_w21 := NOT gvl.Group_01_Axis_11;
gvl.Group_01_Axis_11_Gear_In R= _w21;
gvl.Group_01_Axis_11_Gear_Out S= _w21;

// NETWORK 44
_w22 := gvl.Group_01_Axis_11;
gvl.Group_01_Axis_11_Gear_In S= _w22;
gvl.Group_01_Axis_11_Gear_Out R= _w22;

// NETWORK 45
_w23 := NOT gvl.Group_01_Axis_12;
gvl.Group_01_Axis_12_Gear_In R= _w23;
gvl.Group_01_Axis_12_Gear_Out S= _w23;

// NETWORK 46
_w24 := gvl.Group_01_Axis_12;
gvl.Group_01_Axis_12_Gear_In S= _w24;
gvl.Group_01_Axis_12_Gear_Out R= _w24;

// NETWORK 47
_w25 := NOT gvl.Group_01_Axis_13;
gvl.Group_01_Axis_13_Gear_In R= _w25;
gvl.Group_01_Axis_13_Gear_Out S= _w25;

// NETWORK 48
_w26 := gvl.Group_01_Axis_13;
gvl.Group_01_Axis_13_Gear_In S= _w26;
gvl.Group_01_Axis_13_Gear_Out R= _w26;

// NETWORK 49
_w27 := NOT gvl.Group_01_Axis_14;
gvl.Group_01_Axis_14_Gear_In R= _w27;
gvl.Group_01_Axis_14_Gear_Out S= _w27;

// NETWORK 50
_w28 := gvl.Group_01_Axis_14;
gvl.Group_01_Axis_14_Gear_In S= _w28;
gvl.Group_01_Axis_14_Gear_Out R= _w28;

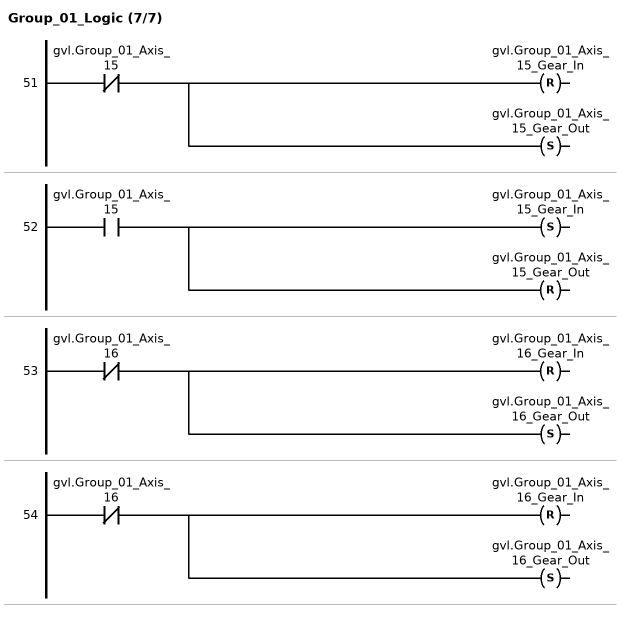
// NETWORK 51
_w29 := NOT gvl.Group_01_Axis_15;
gvl.Group_01_Axis_15_Gear_In R= _w29;
gvl.Group_01_Axis_15_Gear_Out S= _w29;

// NETWORK 52
_w30 := gvl.Group_01_Axis_15;
gvl.Group_01_Axis_15_Gear_In S= _w30;
gvl.Group_01_Axis_15_Gear_Out R= _w30;

// NETWORK 53
_w31 := NOT gvl.Group_01_Axis_16;
gvl.Group_01_Axis_16_Gear_In R= _w31;
gvl.Group_01_Axis_16_Gear_Out S= _w31;

// NETWORK 54
_w32 := NOT gvl.Group_01_Axis_16;
gvl.Group_01_Axis_16_Gear_In R= _w32;
gvl.Group_01_Axis_16_Gear_Out S= _w32;

END_PROGRAM

// ---- POUs/Group_02_Function_Blocks.TcPOU
PROGRAM Group_02_Function_Blocks
VAR
END_VAR

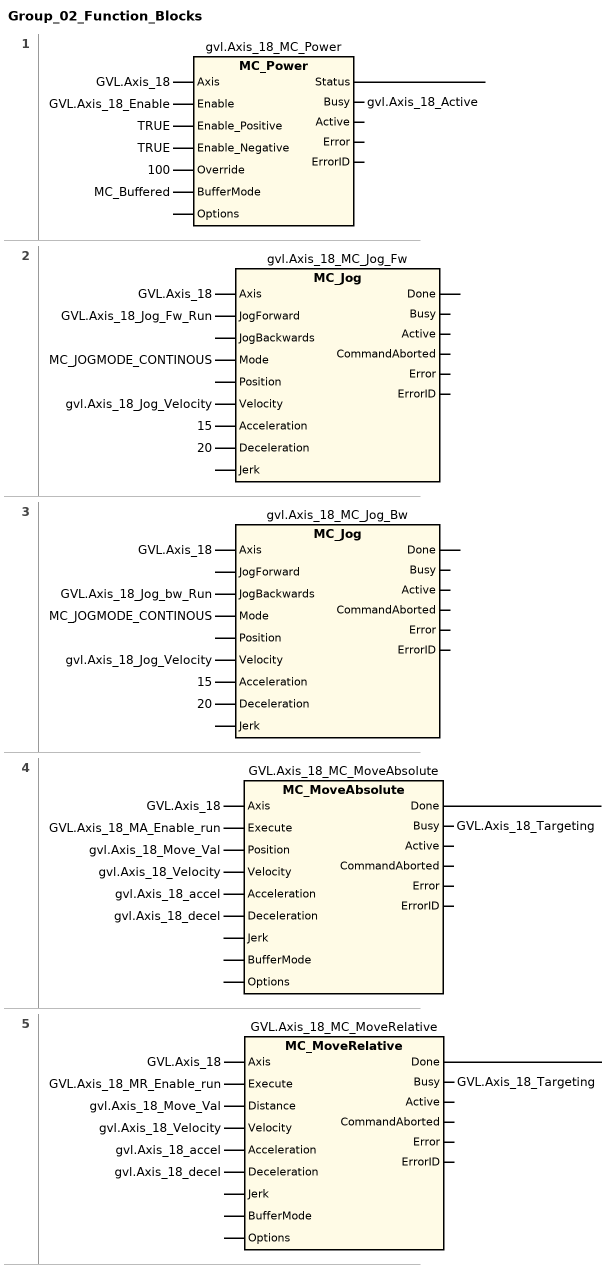
// NETWORK 1
gvl.Axis_18_MC_Power(
    Axis := GVL.Axis_18,
    Enable := GVL.Axis_18_Enable,
    Enable_Positive := TRUE,
    Enable_Negative := TRUE,
    Override := 100,
    BufferMode := MC_Buffered,
    Busy => gvl.Axis_18_Active); // MC_Power

// NETWORK 2
gvl.Axis_18_MC_Jog_Fw(
    Axis := GVL.Axis_18,
    JogForward := GVL.Axis_18_Jog_Fw_Run,
    Mode := MC_JOGMODE_CONTINOUS,
    Velocity := gvl.Axis_18_Jog_Velocity,
    Acceleration := 15,
    Deceleration := 20); // MC_Jog

// NETWORK 3
gvl.Axis_18_MC_Jog_Bw(
    Axis := GVL.Axis_18,
    JogBackwards := GVL.Axis_18_Jog_bw_Run,
    Mode := MC_JOGMODE_CONTINOUS,
    Velocity := gvl.Axis_18_Jog_Velocity,
    Acceleration := 15,
    Deceleration := 20); // MC_Jog

// NETWORK 4
GVL.Axis_18_MC_MoveAbsolute(
    Axis := GVL.Axis_18,
    Execute := GVL.Axis_18_MA_Enable_run,
    Position := gvl.Axis_18_Move_Val,
    Velocity := gvl.Axis_18_Velocity,
    Acceleration := gvl.Axis_18_accel,
    Deceleration := gvl.Axis_18_decel,
    Busy => GVL.Axis_18_Targeting); // MC_MoveAbsolute

// NETWORK 5
GVL.Axis_18_MC_MoveRelative(
    Axis := GVL.Axis_18,
    Execute := GVL.Axis_18_MR_Enable_run,
    Distance := gvl.Axis_18_Move_Val,
    Velocity := gvl.Axis_18_Velocity,
    Acceleration := gvl.Axis_18_accel,
    Deceleration := gvl.Axis_18_decel,
    Busy => GVL.Axis_18_Targeting); // MC_MoveRelative

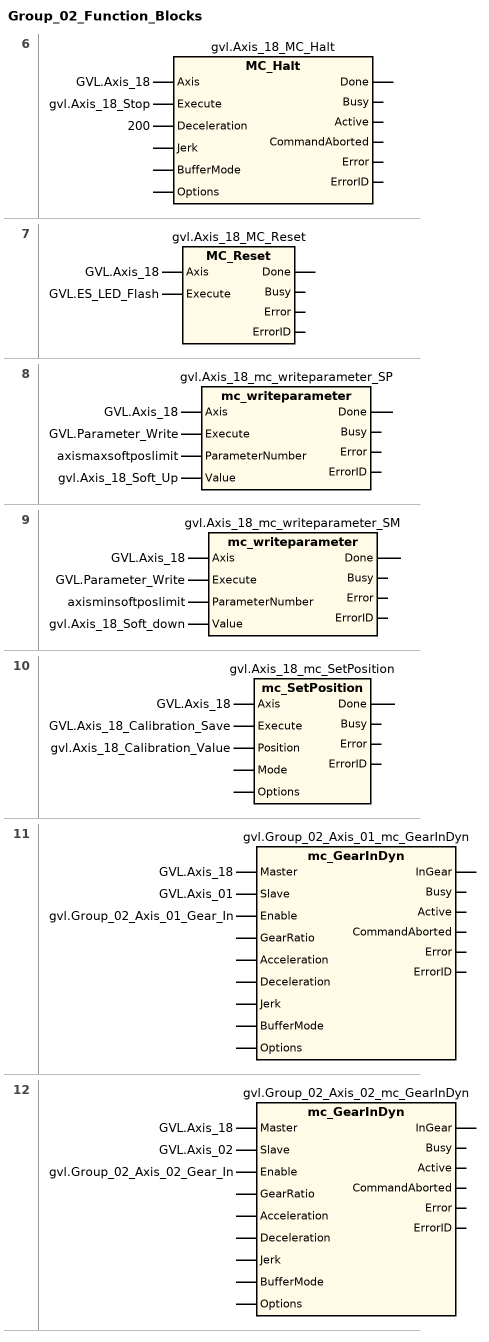
// NETWORK 6
gvl.Axis_18_MC_Halt(Axis := GVL.Axis_18, Execute := gvl.Axis_18_Stop, Deceleration := 200); // MC_Halt

// NETWORK 7
gvl.Axis_18_MC_Reset(Axis := GVL.Axis_18, Execute := GVL.ES_LED_Flash); // MC_Reset

// NETWORK 8
gvl.Axis_18_mc_writeparameter_SP(
    Axis := GVL.Axis_18,
    Execute := GVL.Parameter_Write,
    ParameterNumber := axismaxsoftposlimit,
    Value := gvl.Axis_18_Soft_Up); // mc_writeparameter

// NETWORK 9
gvl.Axis_18_mc_writeparameter_SM(
    Axis := GVL.Axis_18,
    Execute := GVL.Parameter_Write,
    ParameterNumber := axisminsoftposlimit,
    Value := gvl.Axis_18_Soft_down); // mc_writeparameter

// NETWORK 10
gvl.Axis_18_mc_SetPosition(
    Axis := GVL.Axis_18,
    Execute := GVL.Axis_18_Calibration_Save,
    Position := gvl.Axis_18_Calibration_Value); // mc_SetPosition

// NETWORK 11
gvl.Group_02_Axis_01_mc_GearInDyn(
    Master := GVL.Axis_18,
    Slave := GVL.Axis_01,
    Enable := gvl.Group_02_Axis_01_Gear_In); // mc_GearInDyn

// NETWORK 12
gvl.Group_02_Axis_02_mc_GearInDyn(
    Master := GVL.Axis_18,
    Slave := GVL.Axis_02,
    Enable := gvl.Group_02_Axis_02_Gear_In); // mc_GearInDyn

